TYPE
    TcoTixonVibro_Control_v_1_x_x EXTENDS TcoTixonGenericControl :
    STRUCT  
      
        {attribute addProperty Name "<#Shot component#> - q7"}
        ShotComponent : BOOL;
      

    END_STRUCT
END_TYPE

(* stored: Version 1.1.0.1, ProductVersion 3.1.4024.12
   DUT TcoTixonVibro_Control_v_1_x_x: Id {11d73fd2-fa46-05ef-0665-c673170a87de} *)
